{attribute 'GeneratedUsingTerminal: EL3312-0000-0018'}
{attribute addProperty BoxType "EL3312-0000-0018"}
{attribute addProperty Id "TC_Inputs_Channel_1AT %I*AI_Standard_Channel_4A3944819TC_Inputs_Channel_2AT %I*AI_Standard_Channel_4A3944819WcStateAT %I*WcState_9091E0EB2InfoDataAT %I*InfoData_94A18F5E2"}
{attribute addProperty CRC "3547687923"}
{attribute addProperty Size "22"}
TYPE EL3312_D3756BF3 EXTENDS EtcSlaveTerminalBase_947E5A46 :
STRUCT
	{attribute addProperty Name "TC_Inputs_Channel_1"}
	TC_Inputs_Channel_1 : AI_Standard_Channel_4A394481;
	{attribute addProperty Name "TC_Inputs_Channel_2"}
	TC_Inputs_Channel_2 : AI_Standard_Channel_4A394481;
	{attribute addProperty Name "WcState"}
	WcState : WcState_9091E0EB;
	{attribute addProperty Name "InfoData"}
	InfoData : InfoData_94A18F5E;
END_STRUCT
END_TYPE

(* stored: Version 1.2.0.0, ProductVersion 3.1.4024.9
   DUT EL3312_D3756BF3: Id {28a52dfb-1781-4766-b1a5-610117ab6b96} *)
